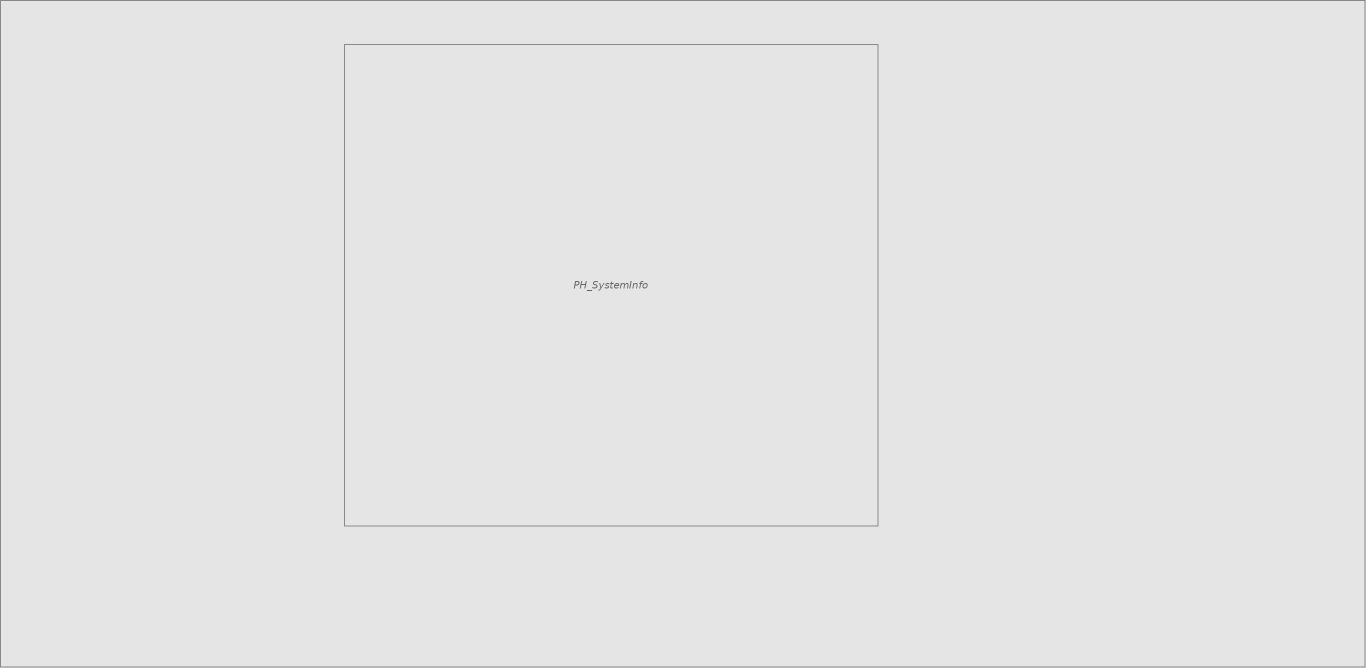
VISUALIZATION V_info  // 1366x668
    TabControl (344,44 534x482)
        shows PH_SystemInfo()
        shows PH_TaskInfo(fbTaskInfo := P_TaskInfo.fbTaskInfo, bReset := P_TaskInfo.fbTaskInfo.bResetVisu)
        shows PH_ControllerInfo(strTargetType := P_ControllerInfo.stDevIdent.strTargetType, strHardwareModel := P_ControllerInfo.stDevIdent.strHardwareModel, strHardwareSerialNo := P_ControllerInfo.stDevIdent.strHardwareSerialNo, strHardwareVersion := P_ControllerInfo.stDevIdent.strHardwareVersion, strHardwareDate := P_ControllerInfo.stDevIdent.strHardwareDate, strHardwareCPU := P_ControllerInfo.stDevIdent.strHardwareCPU, strImageDevice := P_ControllerInfo.stDevIdent.strImageDevice, strImageVersion := P_ControllerInfo.stDevIdent.strImageVersion, strImageLevel := P_ControllerInfo.stDevIdent.strImageLevel, strImageOsName := P_ControllerInfo.stDevIdent.strImageOsName, strImageOsVersion := P_ControllerInfo.stDevIdent.strImageOsVersion, strTwinCATVersion := P_ControllerInfo.stDevIdent.strTwinCATVersion, strTwinCATRevision := P_ControllerInfo.stDevIdent.strTwinCATRevision, strTwinCATBuild := P_ControllerInfo.stDevIdent.strTwinCATBuild, strTwinCATLevel := P_ControllerInfo.stDevIdent.strTwinCATLevel, strAmsNetId := P_ControllerInfo.stDevIdent.strAmsNetId, arrDevIdent := P_ControllerInfo.arrDevIdent, wDeviceInfo := GVL_HMI.wDeviceInfo, iSelectedRow := P_ControllerInfo.iSelectedRow)
        [0]: TabTitle=System Info
        [1]: TabTitle=Task Info
        [2]: TabTitle=Device Info
END_VISUALIZATION

(* stored: Version 1.1.0.1, ProductVersion 3.1.4024.3
   Visu V_info: Id {1d6ab1fa-58de-4a8e-88bd-413c4228b1a6} *)
